// TIA Portal project "Inversión de giro de motor temporizado" (V16)

(* hardware
DEVICE "S7-1200 station_1"  S7-1200 Station
   slot 0: "Rack_0"  S7-1200 Rack  Rack  V1.0
   slot 1: "PLC desconectado"  CPU 1214C DC/DC/DC  6ES7 214-1AG40-0XB0  V4.0
*)

// ===== PLC "PLC desconectado"  CPU 1214C DC/DC/DC =====

VAR_GLOBAL   // PLC tag table "Tabla de variables estándar"
   ""START"" AT %I0.0 : Bool;
   ""STOP"" AT %I0.1 : Bool;
   ""M_Horario"" AT %Q0.0 : Bool;
   ""M_Antihorario"" AT %Q0.1 : Bool;
   ""Espera"" AT %Q0.2 : Bool;
   ""EsperaFinal"" AT %Q0.3 : Bool;
   ""Final"" AT %Q0.4 : Bool;
   ""Libre"" AT %Q0.5 : Bool;
END_VAR